// Widens any numeric value to LREAL so ordering comparisons can be written once
// instead of per type.
//
// Returns ST_NumericValue rather than a value plus an output parameter.
// IsNumeric is FALSE for strings, structs, arrays and anything else with no
// ordering - the caller reports a TypeMismatch rather than comparing rubbish.
//
// LREAL carries 53 bits of mantissa, so LINT and ULINT values beyond 2^53 lose
// precision here. That matters for AssertGreater and AssertLess at extreme
// magnitudes and nowhere else; equality never goes through this path.
FUNCTION TestValueAsLReal : ST_NumericValue
VAR_INPUT
	Value : ANY;
END_VAR

VAR
	Unsigned : ULINT;
	Signed8	 : SINT;
	Signed16 : INT;
	Signed32 : DINT;
	Signed64 : LINT;
	Real32	 : REAL;
	Real64	 : LREAL;
END_VAR

TestValueAsLReal.Value	   := 0.0;
TestValueAsLReal.IsNumeric := TRUE;

CASE Value.TypeClass OF

	__SYSTEM.TYPE_CLASS.TYPE_BYTE,	__SYSTEM.TYPE_CLASS.TYPE_USINT,
	__SYSTEM.TYPE_CLASS.TYPE_WORD,	__SYSTEM.TYPE_CLASS.TYPE_UINT,
	__SYSTEM.TYPE_CLASS.TYPE_DWORD, __SYSTEM.TYPE_CLASS.TYPE_UDINT,
	__SYSTEM.TYPE_CLASS.TYPE_LWORD, __SYSTEM.TYPE_CLASS.TYPE_ULINT:
		MEMCPY(ADR(Unsigned), Value.pValue, TO_UDINT(Value.diSize));
		TestValueAsLReal.Value := TO_LREAL(Unsigned);

	__SYSTEM.TYPE_CLASS.TYPE_SINT:
		MEMCPY(ADR(Signed8), Value.pValue, TO_UDINT(Value.diSize));
		TestValueAsLReal.Value := TO_LREAL(Signed8);

	__SYSTEM.TYPE_CLASS.TYPE_INT:
		MEMCPY(ADR(Signed16), Value.pValue, TO_UDINT(Value.diSize));
		TestValueAsLReal.Value := TO_LREAL(Signed16);

	__SYSTEM.TYPE_CLASS.TYPE_DINT:
		MEMCPY(ADR(Signed32), Value.pValue, TO_UDINT(Value.diSize));
		TestValueAsLReal.Value := TO_LREAL(Signed32);

	__SYSTEM.TYPE_CLASS.TYPE_LINT:
		MEMCPY(ADR(Signed64), Value.pValue, TO_UDINT(Value.diSize));
		TestValueAsLReal.Value := TO_LREAL(Signed64);

	__SYSTEM.TYPE_CLASS.TYPE_REAL:
		MEMCPY(ADR(Real32), Value.pValue, TO_UDINT(Value.diSize));
		TestValueAsLReal.Value := TO_LREAL(Real32);

	__SYSTEM.TYPE_CLASS.TYPE_LREAL:
		MEMCPY(ADR(Real64), Value.pValue, TO_UDINT(Value.diSize));
		TestValueAsLReal.Value := Real64;

ELSE
	TestValueAsLReal.IsNumeric := FALSE;
END_CASE

END_FUNCTION

(* stored: Version 1.1.0.1, ProductVersion 3.1.4026.0
   POU TestValueAsLReal: Id {022dc952-906c-444f-85a9-410ef1ea8c0e}, SpecialFunc None *)
